KUKA KRL data list: TDefault.dat

&ACCESS RV2
DEFDAT TDefault
   INT  I,J,k
ENDDAT
